VAR_IN_OUT
	awBusDataToVTEM 				: ARRAY [0..2] OF WORD; 	(* 6 bytes of process data sent to the Motion Terminal *)	
END_VAR

VAR_INPUT
	xExecute 						: BOOL; 					(* has to be set to TRUE for a download and to FALSE to reset the function block after a download *)
		                    		
	iParameterSet					: INT := 1; 				(* the parameter set to be written to, 1 by default *)
	
	// system parameters
		iTubingLengthAt2 			: INT; 						(* length of the tubing connected to outlet port 2 of the valve [1 digit = 1 mm] *)
		iTubingLengthAt4 			: INT;						(* length of the tubing connected to outlet port 4 of the valve [1 digit = 1 mm] *)
		iTubingInnerDiameterAt2 	: INT;  					(* inner diameter of the tubing connected to outlet port 2 of the valve [1 digit = 0.01 mm] *)
		iTubingInnerDiameterAt4 	: INT;						(* inner diameter of the tubing connected to outlet port 4 of the valve [1 digit = 0.01 mm] *)
		iVolumeAt2 					: INT; 						(* size/capacity of the volume connected to outlet port 2 of the valve [1 digit = 0.001 l] *)
	 	iVolumeAt4 					: INT;						(* size/capacity of the volume connected to outlet port 4 of the valve [1 digit = 0.001 l] *)
		iInPortRetracted_optional	: INT;						// Sensor port for detection of end position at pressurisation of outlet port 2 (retracted), value is number of the slot (beginning from 0) * 10 + number of the port
		iInPortAdvanced_optional	: INT;						// Sensor port for detection of end position at pressurisation of outlet port 4 (advanced), value is number of the slot (beginning from 0) * 10 + number of the port
    
	// application parameters
		iPressureRiseAt2 			: INT; 						(* maximum pressure rise at outlet port 2 [1 digit = 0.01 bar/s] *)
		iPressureRiseAt4 			: INT;						(* maximum pressure rise at outlet port 4 [1 digit = 0.01 bar/s] *)
END_VAR

VAR_OUTPUT
	iResponse 						: eTransferResponse; 		(* returns the status of the execution of the download process *)
	sCurrentValue 					: STRING; 					(* indicates which value of the array is currently treated (necessary to evaluate in case of error messages) *)
	xDownloadDone 					: BOOL; 					(* indicates whether the download was successful *)
	xDownloadError 					: BOOL := FALSE; 			(* indicates whether an error occurred during the transfer *)
END_VAR

VAR
	aTransferPackages				: ARRAY [0..100] OF stTransferPackage;
	fbdownloadMultipleParameters 	: FB_Download_Multiple_Parameters;
	iCurrentValue					: INT;
	fbWriteValueToWord 				: FB_Write_Value_To_Word;
END_VAR

(*****************************************************************************************************

Festo SE & Co. KG, Esslingen
Copyright (c) 2018. All rights reserved.

Product:            Motion Terminal VTEM
Description:        Function block to download the parameters for Motion App 4 to the Motion Terminal

Object version:     2.00
Last change:        2019-03
======================================================================================================
                                       H I S T O R Y
======================================================================================================
Version:            2.00
Date:               2019-03
Change/Activity:    - added parameters for the sensor port mapping (#2256294)
                    - changed awBusDataToVTEM into VAR_IN_OUT (#2368965)
Release:            3.5.7.230 (CODESYS 3.5.7.2, Lib version 3.0)
Author:             JEBU
------------------------------------------------------------------------------------------------------
Version:            1.00
Date:               2017
Change/Activity:    - created
Release:            3.5.7.220
Author:             HLBG
======================================================================================================

*****************************************************************************************************)

// write the Motion App specific parameters into the struct
	//iTubingLengthAt2
		aTransferPackages[0].iChannel := iParameterSet;
		aTransferPackages[0].iAddressedTarget := 4;
		aTransferPackages[0].iIndex := 12;
		aTransferPackages[0].iTransferValue := iTubingLengthAt2;
	
	//iTubingLengthAt4
		aTransferPackages[1].iChannel := iParameterSet;
		aTransferPackages[1].iAddressedTarget := 4;
		aTransferPackages[1].iIndex := 13;
		aTransferPackages[1].iTransferValue := iTubingLengthAt4;
	
	//iTubingInnerDiameterAt2
		aTransferPackages[2].iChannel := iParameterSet;
		aTransferPackages[2].iAddressedTarget := 4;
		aTransferPackages[2].iIndex := 14;
		aTransferPackages[2].iTransferValue := iTubingInnerDiameterAt2;
	
	//iTubingInnerDiameterAt4
		aTransferPackages[3].iChannel := iParameterSet;
		aTransferPackages[3].iAddressedTarget := 4;
		aTransferPackages[3].iIndex := 15;
		aTransferPackages[3].iTransferValue := iTubingInnerDiameterAt4;
	
	//iVolumeAt2
		aTransferPackages[4].iChannel := iParameterSet;
		aTransferPackages[4].iAddressedTarget := 4;
		aTransferPackages[4].iIndex := 40;
		aTransferPackages[4].iTransferValue := iVolumeAt2;
	
	//iVolumeAt4
		aTransferPackages[5].iChannel := iParameterSet;
		aTransferPackages[5].iAddressedTarget := 4;
		aTransferPackages[5].iIndex := 41;
		aTransferPackages[5].iTransferValue := iVolumeAt4;
	
	//iPressureRiseAt2
		aTransferPackages[6].iChannel := iParameterSet;
		aTransferPackages[6].iAddressedTarget := 4;
		aTransferPackages[6].iIndex := 182;
		aTransferPackages[6].iTransferValue := iPressureRiseAt2;
	
	//iPressureRiseAt4
		aTransferPackages[7].iChannel := iParameterSet;
		aTransferPackages[7].iAddressedTarget := 4;
		aTransferPackages[7].iIndex := 183;
		aTransferPackages[7].iTransferValue := iPressureRiseAt4;
	
	//iInPortRetract_optional
		aTransferPackages[8].iChannel := iParameterSet;
		aTransferPackages[8].iAddressedTarget := 4;
		aTransferPackages[8].iIndex := 70;
		aTransferPackages[8].iTransferValue := iInPortRetracted_optional;
	
	//iInPortAdvanced_optional
		aTransferPackages[9].iChannel := iParameterSet;
		aTransferPackages[9].iAddressedTarget := 4;
		aTransferPackages[9].iIndex := 71;
		aTransferPackages[9].iTransferValue := iInPortAdvanced_optional;
	
	// define end of parameter list to be downloaded by setting all variables to 0 (end criterion for FB_Download_Multiple_Parameters)
		aTransferPackages[10].iChannel := 0;
		aTransferPackages[10].iAddressedTarget := 0;
		aTransferPackages[10].iIndex := 0;
		aTransferPackages[10].iTransferValue := 0;


// pre-check of the value for the parameter set
	IF xExecute = TRUE AND (iParameterSet < 1 OR iParameterSet > 5) THEN		// invalid input for the parameter set
		xDownloadDone := FALSE; 
		xDownloadError := TRUE; 
		iResponse := eTransferResponse.invalid_ParameterSet; 
		iCurrentValue := 0; 
		// send command 'stop'
		fbWriteValueToWord(iValue := 61, iStartBit := 0, iEndBit := 5, wDataWord := awBusDataToVTEM[0]); 			// ValveMode = 61
		fbWriteValueToWord(iValue := 0, iStartBit := 6, iEndBit := 15, wDataWord := awBusDataToVTEM[0]); 			// (empty)
		awBusDataToVTEM[1] := 0; 
		awBusDataToVTEM[2] := 0; 
		
	ELSE	
		// call the function block for multiple parameter download
			fbdownloadMultipleParameters(	xExecute := xExecute,
											awBusDataFromVTEM := awBusDataFromVTEM,
											aTransferPackages := aTransferPackages, 
											awBusDataToVTEM := awBusDataToVTEM,
											xDownloadDone => xDownloadDone,
											xDownloadError => xDownloadError,
											iResponse => iResponse,
											iCurrentValue => iCurrentValue);
	END_IF
	

// The current value output is needed if there is any invalid value in order to address it correctly.
// As the user doesn't work with indices in this function block, the current value is transformed to a string holding the name of the parameter.
	CASE iCurrentValue OF
		0: sCurrentValue := 'iTubingLengthAt2';
		1: sCurrentValue := 'iTubingLengthAt4';
		2: sCurrentValue := 'iTubingInnerDiameterAt2';
		3: sCurrentValue := 'iTubingInnerDiameterAt4';
		4: sCurrentValue := 'iVolumeAt2';
		5: sCurrentValue := 'iVolumeAt4';
		6: sCurrentValue := 'iPressureRiseAt2';
		7: sCurrentValue := 'iPressureRiseAt4';
		8: sCurrentValue := 'iInPortRetract_optional';
		9: sCurrentValue := 'iInPortAdvanced_optional';
		10: sCurrentValue := 'AllParametersWritten';
	END_CASE

END_FUNCTION_BLOCK

// Transfermode/specific_MA_config/FB_Write_config_MA_11
/// This function block can be used to download the configuration of Motion App 11 ("Soft stop").
/// The specific parameters of this Motion App are the inputs of this FB and can be defined by the user. 
/// The function block uses the transfer mode to write this configuration to the Motion Terminal
/// and indicates the state of the download process.

FUNCTION_BLOCK FB_Write_config_MA_11
VAR_INPUT
	awBusDataFromVTEM 				: ARRAY [0..2] OF WORD;		(* 6 bytes of process data received from the Motion Terminal *)
END_VAR

VAR_IN_OUT
	awBusDataToVTEM					: ARRAY [0..2] OF WORD; 	(* 6 bytes of process data sent to the Motion Terminal *)
END_VAR

VAR_INPUT
	xExecute 						: BOOL; 					(* has to be set to TRUE for a download and to FALSE to reset the function block after a download *)
	
	iParameterSet					: INT := 1; 				(* the parameter set to be written to, 1 by default *)
	
	// system parameters
		iDriveType 					: INT;						(* type of the drive/cylinder/... that is to be operated by the valve ->  see list of drive types *)
	 	iDriveStroke 				: INT; 						(* stroke of the drive/cylinder/... that is to be operated by the valve [1 digit = 1 mm for linear drives, 1 digit = 1° for rotary drives] *)
		iInstallationPositionDrive 	: INT;  	 				(* inclination of the cylinder with reference to a horizontal installation position [1 digit = 0.01°, positive values = advancing upwards] *)
		iInPortRetracted			: INT;						// Sensor port for detection of end position at pressurisation of outlet port 2 (retracted), value is number of the slot (beginning from 0) * 10 + number of the port
		iInPortAdvanced				: INT;						// Sensor port for detection of end position at pressurisation of outlet port 4 (advanced), value is number of the slot (beginning from 0) * 10 + number of the port
	
	// application parameters                               	
	 	iLoadAdvancing 				: INT := 0; 				(* mass that is to be moved by the drive when advancing ((4) pressurised) [1 digit = 0.01 kg] *)
		iLoadRetracting 			: INT := 0;					(* mass that is to be moved by the drive when retracting ((2) pressurised) [1 digit = 0.01 kg] *)

END_VAR

VAR_OUTPUT                                                  	
	iResponse 						: eTransferResponse; 		(* returns the status of the execution of the download process *)
	sCurrentValue 					: STRING; 					(* indicates which value of the array is currently treated (necessary to evaluate in case of error messages) *)
	xDownloadDone 					: BOOL; 					(* indicates whether the download was successful *)
	xDownloadError 					: BOOL := FALSE; 			(* indicates whether an error occurred during the transfer *)
END_VAR

VAR
	aTransferPackages				: ARRAY [0..100] OF stTransferPackage;
	fbdownloadMultipleParameters 	: FB_Download_Multiple_Parameters;
	iCurrentValue					: INT;
	fbWriteValueToWord 				: FB_Write_Value_To_Word;
END_VAR

(*****************************************************************************************************

Festo SE & Co. KG, Esslingen
Copyright (c) 2018. All rights reserved.

Product:            Motion Terminal VTEM
Description:        Function block to download the parameters for Motion App 11 to the Motion Terminal

Object version:     2.01
Last change:        2019-03
======================================================================================================
                                       H I S T O R Y
======================================================================================================
Version:            2.01
Date:               2019-03
Change/Activity:    - sensor port mapping parameters (#2397241)
Release:            3.5.7.231 (CODESYS 3.5.7.2, Lib version 3.1)
Author:             JEBU
------------------------------------------------------------------------------------------------------
Version:            2.00
Date:               2019-03
Change/Activity:    - added parameters for the sensor port mapping (#2256294)
                    - removed tuning parameters (#2374189)
                    - changed awBusDataToVTEM into VAR_IN_OUT (#2368965)
Release:            3.5.7.230 (CODESYS 3.5.7.2, Lib version 3.0)
Author:             JEBU
------------------------------------------------------------------------------------------------------
Version:            1.01
Date:               2018-08
Change/Activity:    - added tuning parameters
Release:            3.5.7.220
Author:             JEBU
------------------------------------------------------------------------------------------------------
Version:            1.00
Date:               2017
Change/Activity:    - created
Release:            not released
Author:             HLBG
======================================================================================================

*****************************************************************************************************)

// write the Motion App specific parameters into the struct
	//iDriveType
		aTransferPackages[0].iChannel := iParameterSet;
		aTransferPackages[0].iAddressedTarget := 11;
		aTransferPackages[0].iIndex := 20;
		aTransferPackages[0].iTransferValue := iDriveType;
		
	//iDriveStroke
		aTransferPackages[1].iChannel := iParameterSet;
		aTransferPackages[1].iAddressedTarget := 11;
		aTransferPackages[1].iIndex := 21;
		aTransferPackages[1].iTransferValue := iDriveStroke;
		
	//iInstallationPositionDrive
		aTransferPackages[2].iChannel := iParameterSet;
		aTransferPackages[2].iAddressedTarget := 11;
		aTransferPackages[2].iIndex := 60;
		aTransferPackages[2].iTransferValue := iInstallationPositionDrive;
		
	//iLoadAdvancing
		aTransferPackages[3].iChannel := iParameterSet;
		aTransferPackages[3].iAddressedTarget := 11;
		aTransferPackages[3].iIndex := 101;
		aTransferPackages[3].iTransferValue := iLoadAdvancing;
		
	//iLoadRetracting
		aTransferPackages[4].iChannel := iParameterSet;
		aTransferPackages[4].iAddressedTarget := 11;
		aTransferPackages[4].iIndex := 100;
		aTransferPackages[4].iTransferValue := iLoadRetracting;
		
	//iInPortRetract
		aTransferPackages[5].iChannel := iParameterSet;
		aTransferPackages[5].iAddressedTarget := 11;
		aTransferPackages[5].iIndex := 75;
		aTransferPackages[5].iTransferValue := iInPortRetracted;
	
	//iInPortRetract
		aTransferPackages[6].iChannel := iParameterSet;
		aTransferPackages[6].iAddressedTarget := 11;
		aTransferPackages[6].iIndex := 76;
		aTransferPackages[6].iTransferValue := iInPortAdvanced;
	
	// define end of parameter list to be downloaded by setting all variables to 0 (end criterion for FB_Download_Multiple_Parameters)
		aTransferPackages[7].iChannel := 0;
		aTransferPackages[7].iAddressedTarget := 0;
		aTransferPackages[7].iIndex := 0;
		aTransferPackages[7].iTransferValue := 0;


// pre-check of the value for the parameter set
	IF xExecute = TRUE AND (iParameterSet < 1 OR iParameterSet > 5) THEN		// invalid input for the parameter set
		xDownloadDone := FALSE; 
		xDownloadError := TRUE; 
		iResponse := eTransferResponse.invalid_ParameterSet; 
		iCurrentValue := 0; 
		// send command 'stop'
		fbWriteValueToWord(iValue := 61, iStartBit := 0, iEndBit := 5, wDataWord := awBusDataToVTEM[0]); 			// ValveMode = 61
		fbWriteValueToWord(iValue := 0, iStartBit := 6, iEndBit := 15, wDataWord := awBusDataToVTEM[0]); 			// (empty)
		awBusDataToVTEM[1] := 0; 
		awBusDataToVTEM[2] := 0; 
		
	ELSE	
		// call the function block for multiple parameter download
			fbdownloadMultipleParameters(	xExecute := xExecute,
											awBusDataFromVTEM := awBusDataFromVTEM,
											aTransferPackages := aTransferPackages, 
											awBusDataToVTEM := awBusDataToVTEM,
											xDownloadDone => xDownloadDone,
											xDownloadError => xDownloadError,
											iResponse => iResponse,
											iCurrentValue => iCurrentValue);
	END_IF
		
	
// The current value output is needed if there is any invalid value in order to address it correctly.
// As the user doesn't work with indices in this function block, the current value is transformed to a string holding the name of the parameter.
	CASE iCurrentValue OF
		0: sCurrentValue := 'iDriveType';
		1: sCurrentValue := 'iDriveStroke';
		2: sCurrentValue := 'iInstallationPositionDrive';
		3: sCurrentValue := 'iLoadAdvancing';
		4: sCurrentValue := 'iLoadRetracting';
		5: sCurrentValue := 'iInPortRetract';
		6: sCurrentValue := 'iInPortAdvanced';
		7: sCurrentValue := 'AllParametersWritten';
	END_CASE

END_FUNCTION_BLOCK

// Transfermode/specific_MA_config/FB_Write_config_MA_12
/// This function block can be used to download the configuration of Motion App 12 ("Leakage diagnostics").
/// The specific parameters of this Motion App are the inputs of this FB and can be defined by the user. 
/// The function block uses the transfer mode to write this configuration to the Motion Terminal
/// and indicates the state of the download process.

FUNCTION_BLOCK FB_Write_config_MA_12
VAR_INPUT
	awBusDataFromVTEM 				: ARRAY [0..2] OF WORD;		(* 6 bytes of process data received from the Motion Terminal *)
END_VAR

VAR_IN_OUT
	awBusDataToVTEM 				: ARRAY [0..2] OF WORD; 	(* 6 bytes of process data sent to the Motion Terminal *)
END_VAR

VAR_INPUT
	xExecute 						: BOOL; 					(* has to be set to TRUE for a download and to FALSE to reset the function block after a download *)
		                                                    	
	iParameterSet					: INT := 1; 				(* the parameter set to be written to, 1 by default *)
	
	// system parameters
		iTubingLengthAt2 			: INT; 						(* length of the tubing connected to outlet port 2 of the valve [1 digit = 1 mm] *)
	 	iTubingLengthAt4 			: INT;						(* length of the tubing connected to outlet port 4 of the valve [1 digit = 1 mm] *)
	 	iTubingInnerDiameterAt2		: INT;  					(* inner diameter of the tubing connected to outlet port 2 of the valve [1 digit = 0.01mm] *)
	 	iTubingInnerDiameterAt4		: INT;						(* inner diameter of the tubing connected to outlet port 4 of the valve [1 digit = 0.01mm] *)
	 	iDriveType 					: INT;						(* type of the drive/cylinder/... that is to be operated by the valve ->  see list of drive types *)
	 	iDriveStroke 				: INT; 						(* stroke of the drive/cylinder/... that is to be operated by the valve [1 digit = 1 mm for linear drives, 1 digit = 1° for rotary drives] *)
		iVolumeAt2 					: INT; 						(* size/capacity of the volume connected to outlet port 2 of the valve [1 digit = 0.001 l] *)
		iVolumeAt4 					: INT;						(* size/capacity of the volume connected to outlet port 4 of the valve [1 digit = 0.001 l] *)
		iInstallationPositionDrive 	: INT;  	 				(* inclination of the cylinder with reference to a horizontal installation position [1 digit = 0.01°, positive values = advancing upwards] *)

	// application parameters                               	
		iLoadRetracting 			: INT;						(* mass that is to be moved by the drive when retracting ((2) pressurised) [1 digit = 0.01 kg] *)
	 	iLoadAdvancing 				: INT; 						(* mass that is to be moved by the drive when advancing ((4) pressurised) [1 digit = 0.01 kg] *)
		iMomentOfInertiaRetracting	: INT;						// Moment of inertia during for swivel drives when retratcting ((2) pressirised) [1 digit = 1 kg cm³]
		iMomentOfInertiaAdvancing	: INT;						// Moment of inertia during for swivel drives when advancing ((4) pressirised) [1 digit = 1 kg cm³]
		iMaxLeakageForStatusGood 	: INT;						(* allowed deviation regarding reference value for status "Good" [1 digit = 0.1 l/h] *)
		iMaxLeakageForStatusWarning : INT;						(* allowed deviation regarding reference value for status "Warning" [1 digit = 0.1 l/h] *)
	 	iMaxLeakageForStatusCritical: INT; 						(* allowed deviation regarding reference value for status "Critical" [1 digit = 0.1 l/h] *)
END_VAR

VAR_OUTPUT                                                  	
	iResponse 						: eTransferResponse;		(* returns the status of the execution of the download process *)
	sCurrentValue 					: STRING; 					(* indicates which value of the array is currently treated (necessary to evaluate in case of error messages) *)
	xDownloadDone 					: BOOL; 					(* indicates whether the download was successful *)
	xDownloadError 					: BOOL := FALSE; 			(* indicates whether an error occurred during the transfer *)
END_VAR

VAR
	aTransferPackages				: ARRAY [0..100] OF stTransferPackage;
	fbdownloadMultipleParameters 	: FB_Download_Multiple_Parameters;
	iCurrentValue					: INT;
	fbWriteValueToWord 				: FB_Write_Value_To_Word;
END_VAR

(*****************************************************************************************************

Festo SE & Co. KG, Esslingen
Copyright (c) 2018. All rights reserved.

Product:            Motion Terminal VTEM
Description:        Function block to download the parameters for Motion App 12 to the Motion Terminal

Object version:     2.01
Last change:        2019-04
======================================================================================================
                                       H I S T O R Y
======================================================================================================
Version:            2.01
Date:               2019-04
Change/Activity:    - added parameters for moment of inertia used for swivel drives (#2307852)
                    - changed awBusDataToVTEM into VAR_IN_OUT (#2368965)
Release:            3.5.7.231 (CODESYS 3.5.7.2, Lib version 3.1)
Author:             JEBU
------------------------------------------------------------------------------------------------------
Version:            1.00
Date:               2017
Change/Activity:    - created
Release:            3.5.7.22 (CODESYS 3.5.7.2, Lib version 2.0)
Author:             HLBG
======================================================================================================

*****************************************************************************************************)

// write the Motion App specific parameters into the struct
	//iTubingLengthAt2
		aTransferPackages[0].iChannel := iParameterSet;
		aTransferPackages[0].iAddressedTarget := 12;
		aTransferPackages[0].iIndex := 12;
		aTransferPackages[0].iTransferValue := iTubingLengthAt2;
		
	//iTubingLengthAt4
		aTransferPackages[1].iChannel := iParameterSet;
		aTransferPackages[1].iAddressedTarget := 12;
		aTransferPackages[1].iIndex := 13;
		aTransferPackages[1].iTransferValue := iTubingLengthAt4;
		
	//iTubingInnerDiameterAt2
		aTransferPackages[2].iChannel := iParameterSet;
		aTransferPackages[2].iAddressedTarget := 12;
		aTransferPackages[2].iIndex := 14;
		aTransferPackages[2].iTransferValue := iTubingInnerDiameterAt2;
		
	//iTubingInnerDiameterAt4
		aTransferPackages[3].iChannel := iParameterSet;
		aTransferPackages[3].iAddressedTarget := 12;
		aTransferPackages[3].iIndex := 15;
		aTransferPackages[3].iTransferValue := iTubingInnerDiameterAt4;
		
	//iDriveType
		aTransferPackages[4].iChannel := iParameterSet;
		aTransferPackages[4].iAddressedTarget := 12;
		aTransferPackages[4].iIndex := 20;
		aTransferPackages[4].iTransferValue := iDriveType;
		
	//iDriveStroke
		aTransferPackages[5].iChannel := iParameterSet;
		aTransferPackages[5].iAddressedTarget := 12;
		aTransferPackages[5].iIndex := 21;
		aTransferPackages[5].iTransferValue := iDriveStroke;
		
	//iVolumeAt2
		aTransferPackages[6].iChannel := iParameterSet;
		aTransferPackages[6].iAddressedTarget := 12;
		aTransferPackages[6].iIndex := 40;
		aTransferPackages[6].iTransferValue := iVolumeAt2;
		
	//iVolumeAt4 
		aTransferPackages[7].iChannel := iParameterSet;
		aTransferPackages[7].iAddressedTarget := 12;
		aTransferPackages[7].iIndex := 41;
		aTransferPackages[7].iTransferValue := iVolumeAt4;
		
	//iInstallationPositionDrive
		aTransferPackages[8].iChannel := iParameterSet;
		aTransferPackages[8].iAddressedTarget := 12;
		aTransferPackages[8].iIndex := 60;
		aTransferPackages[8].iTransferValue := iInstallationPositionDrive;
		
	//iLoadRetracting
		aTransferPackages[9].iChannel := iParameterSet;
		aTransferPackages[9].iAddressedTarget := 12;
		aTransferPackages[9].iIndex := 100;
		aTransferPackages[9].iTransferValue := iLoadRetracting;
		
	//iLoadAdvancing
		aTransferPackages[10].iChannel := iParameterSet;
		aTransferPackages[10].iAddressedTarget := 12;
		aTransferPackages[10].iIndex := 101;
		aTransferPackages[10].iTransferValue := iLoadAdvancing;
		
	//iMomentOfInertiaRetracting
		aTransferPackages[11].iChannel := iParameterSet;
		aTransferPackages[11].iAddressedTarget := 12;
		aTransferPackages[11].iIndex := 102;
		aTransferPackages[11].iTransferValue := iMomentOfInertiaRetracting;
	
	//iMomentOfInertiaAdvancing
		aTransferPackages[12].iChannel := iParameterSet;
		aTransferPackages[12].iAddressedTarget := 12;
		aTransferPackages[12].iIndex := 103;
		aTransferPackages[12].iTransferValue := iMomentOfInertiaAdvancing;

	//iMaxLeakageForStatusGood
		aTransferPackages[13].iChannel := iParameterSet;
		aTransferPackages[13].iAddressedTarget := 12;
		aTransferPackages[13].iIndex := 200;
		aTransferPackages[13].iTransferValue := iMaxLeakageForStatusGood;
		
	//iMaxLeakageForStatusWarning
		aTransferPackages[14].iChannel := iParameterSet;
		aTransferPackages[14].iAddressedTarget := 12;
		aTransferPackages[14].iIndex := 201;
		aTransferPackages[14].iTransferValue := iMaxLeakageForStatusWarning;
		
	//iMaxLeakageForStatusCritical
		aTransferPackages[15].iChannel := iParameterSet;
		aTransferPackages[15].iAddressedTarget := 12;
		aTransferPackages[15].iIndex := 202;
		aTransferPackages[15].iTransferValue := iMaxLeakageForStatusCritical;
	
	// define end of parameter list to be downloaded by setting all variables to 0 (end criterion for FB_Download_Multiple_Parameters)
		aTransferPackages[16].iChannel := 0;
		aTransferPackages[16].iAddressedTarget := 0;
		aTransferPackages[16].iIndex := 0;
		aTransferPackages[16].iTransferValue := 0;


// pre-check of the value for the parameter set
	IF xExecute = TRUE AND (iParameterSet < 1 OR iParameterSet > 5) THEN		// invalid input for the parameter set
		xDownloadDone := FALSE; 
		xDownloadError := TRUE; 
		iResponse := eTransferResponse.invalid_ParameterSet; 
		iCurrentValue := 0; 
		// send command 'stop'
		fbWriteValueToWord(iValue := 61, iStartBit := 0, iEndBit := 5, wDataWord := awBusDataToVTEM[0]); 			// ValveMode = 61
		fbWriteValueToWord(iValue := 0, iStartBit := 6, iEndBit := 15, wDataWord := awBusDataToVTEM[0]); 			// (empty)
		awBusDataToVTEM[1] := 0; 
		awBusDataToVTEM[2] := 0; 
		
	ELSE	
		// call the function block for multiple parameter download
			fbdownloadMultipleParameters(	xExecute := xExecute,
											awBusDataFromVTEM := awBusDataFromVTEM,
											aTransferPackages := aTransferPackages, 
											awBusDataToVTEM := awBusDataToVTEM,
											xDownloadDone => xDownloadDone,
											xDownloadError => xDownloadError,
											iResponse => iResponse,
											iCurrentValue => iCurrentValue);
	END_IF
		
	
// The current value output is needed if there is any invalid value in order to address it correctly.
// As the user doesn't work with indices in this function block, the current value is transformed to a string holding the name of the parameter.
	CASE iCurrentValue OF
		0: sCurrentValue := 'iTubingLengthAt2';
		1: sCurrentValue := 'iTubingLengthAt4';
		2: sCurrentValue := 'iTubingInnerDiameterAt2';
		3: sCurrentValue := 'iTubingInnerDiameterAt4';
		4: sCurrentValue := 'iDriveType';
		5: sCurrentValue := 'iDriveStroke';
		6: sCurrentValue := 'iVolumeAt2';
		7: sCurrentValue := 'iVolumeAt4';
		8: sCurrentValue := 'iInstallationPositionDrive';
		9: sCurrentValue := 'iLoadRetracting';
		10: sCurrentValue := 'iLoadAdvancing';
		11: sCurrentValue := 'iMomentOfInertiaRetracting';
		12: sCurrentValue := 'iMomentOfInertiaAdvancing';
		13: sCurrentValue := 'iMaxLeakageForStatusGood';
		14: sCurrentValue := 'iMaxLeakageForStatusWarning';
		15: sCurrentValue := 'iMaxLeakageForStatusCritical';
		16: sCurrentValue := 'AllParametersWritten';
	END_CASE

END_FUNCTION_BLOCK

// StateInterpreter/FB_StateInterpreter_MA_02
/// The variable "byActualAppState" is an output of the FB_ValveControl that is used differently in each Motion App.
/// This function block interprets the "AppState" output of the FB_ValveControl if Motion App 2 ("Proportional directional control valve") is running.
/// The Motion App specific values are derived from the "byActualAppState".

FUNCTION_BLOCK FB_StateInterpreter_MA_02
VAR_INPUT
	byActualAppState 			: BYTE; 	(* output of the FB_ValveControl *)
END_VAR
VAR_OUTPUT
	xRetractedEndPos_optional	: BOOL;  	(* only if digital sensors are installed (optional): indicates whether the retracted end position was reached (after outlet port 2 is pressurised) *)
	xAdvancedEndPos_optional	: BOOL;  	(* only if digital sensors are installed (optional): indicates whether the advanced end position was reached (after outlet port 4 is pressurised) *)
	xWarning					: BOOL; 	(* indicates whether there is a warning returned by the Motion App *)
END_VAR
VAR
	fbReadBitsFromByte			: FB_Read_Bits_From_Byte;
	byRetractedEndPos			: BYTE;
	byAdvancedEndPos			: BYTE;
	byWarning					: BYTE;
END_VAR

(*****************************************************************************************************

Festo SE & Co. KG, Esslingen
Copyright (c) 2018. All rights reserved.

Product:            Motion Terminal VTEM
Description:        Function block for interpreting the app state of Motion App 2

Object version:     1.00
Last change:        2017
======================================================================================================
                                       H I S T O R Y
======================================================================================================
Version:            1.00
Date:               2017
Change/Activity:    - created
Release:            3.5.7.220
Author:             HLBG
======================================================================================================

*****************************************************************************************************)

// read the Motion App specific values from the ActualAppState byte
fbReadBitsFromByte(byData := byActualAppState, iStartBit := 0, iEndBit := 0, byValue => byRetractedEndPos);
xRetractedEndPos_optional :=  BYTE_TO_BIT(byRetractedEndPos);

fbReadBitsFromByte(byData := byActualAppState, iStartBit := 2, iEndBit := 2, byValue => byAdvancedEndPos); 
xAdvancedEndPos_optional :=  BYTE_TO_BIT(byAdvancedEndPos);

fbReadBitsFromByte(byData := byActualAppState, iStartBit := 7, iEndBit := 7, byValue => byWarning);
xWarning := BYTE_TO_BIT(byWarning);

END_FUNCTION_BLOCK

// StateInterpreter/FB_StateInterpreter_MA_03
/// The variable "byActualAppState" is an output of the FB_ValveControl that is used differently in each Motion App.
/// This function block interprets the "AppState" output of the FB_ValveControl if Motion App 3 ("Proportional pressure regulation") is running.
/// The Motion App specific values are derived from the "byActualAppState".

FUNCTION_BLOCK FB_StateInterpreter_MA_03
VAR_INPUT
	byActualAppState 			: BYTE; 	(* output of the FB_ValveControl *)
END_VAR
VAR_OUTPUT
	xRetractedEndPos_optional	: BOOL;  	(* only if digital sensors are installed (optional): indicates whether the retracted end position was reached (after outlet port 2 is pressurised) *)
	xAdvancedEndPos_optional	: BOOL;  	(* only if digital sensors are installed (optional): indicates whether the advanced end position was reached (after outlet port 4 is pressurised) *)
	xWarning					: BOOL; 	(* indicates whether there is a warning returned by the Motion App *)
END_VAR
VAR
	fbReadBitsFromByte			: FB_Read_Bits_From_Byte;
	byRetractedEndPos			: BYTE;
	byAdvancedEndPos			: BYTE;
	byWarning					: BYTE;
END_VAR

(*****************************************************************************************************

Festo SE & Co. KG, Esslingen
Copyright (c) 2018. All rights reserved.

Product:            Motion Terminal VTEM
Description:        Function block for interpreting the app state of Motion App 3

Object version:     1.00
Last change:        2017
======================================================================================================
                                       H I S T O R Y
======================================================================================================
Version:            1.00
Date:               2017
Change/Activity:    - created
Release:            3.5.7.220
Author:             HLBG
======================================================================================================

*****************************************************************************************************)

// read the Motion App specific values from the ActualAppState byte
fbReadBitsFromByte(byData := byActualAppState, iStartBit := 0, iEndBit := 0, byValue => byRetractedEndPos);
xRetractedEndPos_optional :=  BYTE_TO_BIT(byRetractedEndPos);

fbReadBitsFromByte(byData := byActualAppState, iStartBit := 2, iEndBit := 2, byValue => byAdvancedEndPos); 
xAdvancedEndPos_optional :=  BYTE_TO_BIT(byAdvancedEndPos);

fbReadBitsFromByte(byData := byActualAppState, iStartBit := 7, iEndBit := 7, byValue => byWarning);
xWarning := BYTE_TO_BIT(byWarning);

END_FUNCTION_BLOCK

// StateInterpreter/FB_StateInterpreter_MA_04
/// The variable "byActualAppState" is an output of the FB_ValveControl that is used differently in each Motion App.
/// This function block interprets the "AppState" output of the FB_ValveControl if Motion App 4 ("Model-based proportional pressure regulation") is running.
/// The Motion App specific values are derived from the "byActualAppState".

FUNCTION_BLOCK FB_StateInterpreter_MA_04
VAR_INPUT
	byActualAppState 			: BYTE; 	(* output of the FB_ValveControl *)
END_VAR
VAR_OUTPUT
	xRetractedEndPos_optional	: BOOL;  	(* only if digital sensors are installed (optional): indicates whether the retracted end position was reached (after outlet port 2 is pressurised) *)
	xAdvancedEndPos_optional	: BOOL;  	(* only if digital sensors are installed (optional): indicates whether the advanced end position was reached (after outlet port 4 is pressurised) *)
	xWarning					: BOOL; 	(* indicates whether there is a warning returned by the Motion App *)
END_VAR
VAR
	fbReadBitsFromByte			: FB_Read_Bits_From_Byte;
	byRetractedEndPos			: BYTE;
	byAdvancedEndPos			: BYTE;
	byWarning					: BYTE;
END_VAR

(*****************************************************************************************************

Festo SE & Co. KG, Esslingen
Copyright (c) 2018. All rights reserved.

Product:            Motion Terminal VTEM
Description:        Function block for interpreting the app state of Motion App 4

Object version:     1.00
Last change:        2017
======================================================================================================
                                       H I S T O R Y
======================================================================================================
Version:            1.00
Date:               2017
Change/Activity:    - created
Release:            3.5.7.220
Author:             HLBG
======================================================================================================

*****************************************************************************************************)

// read the Motion App specific values from the ActualAppState byte
fbReadBitsFromByte(byData := byActualAppState, iStartBit := 0, iEndBit := 0, byValue => byRetractedEndPos);
xRetractedEndPos_optional :=  BYTE_TO_BIT(byRetractedEndPos);

fbReadBitsFromByte(byData := byActualAppState, iStartBit := 2, iEndBit := 2, byValue => byAdvancedEndPos); 
xAdvancedEndPos_optional :=  BYTE_TO_BIT(byAdvancedEndPos);

fbReadBitsFromByte(byData := byActualAppState, iStartBit := 7, iEndBit := 7, byValue => byWarning);
xWarning := BYTE_TO_BIT(byWarning);

END_FUNCTION_BLOCK

// StateInterpreter/FB_StateInterpreter_MA_05
/// The variable "byActualAppState" is an output of the FB_ValveControl that is used differently in each Motion App.
/// This function block interprets the "AppState" output of the FB_ValveControl if Motion App 5 ("Supply and exhaust air flow control") is running.
/// The Motion App specific values are derived from the "byActualAppState".

FUNCTION_BLOCK FB_StateInterpreter_MA_05
VAR_INPUT
	byActualAppState 			: BYTE; 	(* output of the FB_ValveControl *)
END_VAR
VAR_OUTPUT
	xRetractedEndPos_optional	: BOOL;  	(* only if digital sensors are installed (optional): indicates whether the retracted end position was reached (after outlet port 2 is pressurised) *)
	xAdvancedEndPos_optional	: BOOL;  	(* only if digital sensors are installed (optional): indicates whether the advanced end position was reached (after outlet port 4 is pressurised) *)
	xWarning					: BOOL; 	(* indicates whether there is a warning returned by the Motion App *)
END_VAR
VAR
	fbReadBitsFromByte			: FB_Read_Bits_From_Byte;
	byRetractedEndPos			: BYTE;
	byAdvancedEndPos			: BYTE;
	byWarning					: BYTE;
END_VAR

(*****************************************************************************************************

Festo SE & Co. KG, Esslingen
Copyright (c) 2018. All rights reserved.

Product:            Motion Terminal VTEM
Description:        Function block for interpreting the app state of Motion App 5 

Object version:     1.00
Last change:        2017
======================================================================================================
                                       H I S T O R Y
======================================================================================================
Version:            1.00
Date:               2017
Change/Activity:    - created
Release:            3.5.7.220
Author:             HLBG
======================================================================================================

*****************************************************************************************************)

// read the Motion App specific values from the ActualAppState byte
fbReadBitsFromByte(byData := byActualAppState, iStartBit := 0, iEndBit := 0, byValue => byRetractedEndPos);
xRetractedEndPos_optional :=  BYTE_TO_BIT(byRetractedEndPos);

fbReadBitsFromByte(byData := byActualAppState, iStartBit := 2, iEndBit := 2, byValue => byAdvancedEndPos); 
xAdvancedEndPos_optional :=  BYTE_TO_BIT(byAdvancedEndPos);

fbReadBitsFromByte(byData := byActualAppState, iStartBit := 7, iEndBit := 7, byValue => byWarning);
xWarning := BYTE_TO_BIT(byWarning);

END_FUNCTION_BLOCK

// StateInterpreter/FB_StateInterpreter_MA_08
/// The variable "byActualAppState" is an output of the FB_ValveControl that is used differently in each Motion App.
/// This function block interprets the "AppState" output of the FB_ValveControl if Motion App 8 ("Selectable pressure level (ECO)") is running.
/// The Motion App specific values are derived from the "byActualAppState".

FUNCTION_BLOCK FB_StateInterpreter_MA_08
VAR_INPUT
	byActualAppState 			: BYTE; 	(* output of the FB_ValveControl *)
END_VAR
VAR_OUTPUT
	xRetractedEndPos_optional	: BOOL;  	(* only if digital sensors are installed (optional): indicates whether the retracted end position was reached (after outlet port 2 is pressurised) *)
	xAdvancedEndPos_optional	: BOOL;  	(* only if digital sensors are installed (optional): indicates whether the advanced end position was reached (after outlet port 4 is pressurised) *)
	xWarning					: BOOL; 	(* indicates whether there is a warning returned by the Motion App *)
END_VAR
VAR
	fbReadBitsFromByte			: FB_Read_Bits_From_Byte;
	byRetractedEndPos			: BYTE;
	byAdvancedEndPos			: BYTE;
	byWarning					: BYTE;
END_VAR

(*****************************************************************************************************

Festo SE & Co. KG, Esslingen
Copyright (c) 2018. All rights reserved.

Product:            Motion Terminal VTEM
Description:        Function block for interpreting the app state of Motion App 8 

Object version:     1.00
Last change:        2017
======================================================================================================
                                       H I S T O R Y
======================================================================================================
Version:            1.00
Date:               2017
Change/Activity:    - created
Release:            3.5.7.220
Author:             HLBG
======================================================================================================

*****************************************************************************************************)

// read the Motion App specific values from the ActualAppState byte
fbReadBitsFromByte(byData := byActualAppState, iStartBit := 0, iEndBit := 0, byValue => byRetractedEndPos);
xRetractedEndPos_optional :=  BYTE_TO_BIT(byRetractedEndPos);

fbReadBitsFromByte(byData := byActualAppState, iStartBit := 2, iEndBit := 2, byValue => byAdvancedEndPos); 
xAdvancedEndPos_optional :=  BYTE_TO_BIT(byAdvancedEndPos);

fbReadBitsFromByte(byData := byActualAppState, iStartBit := 7, iEndBit := 7, byValue => byWarning);
xWarning := BYTE_TO_BIT(byWarning);

END_FUNCTION_BLOCK

// Transfermode/specific_MA_config/FB_Write_config_MA_02
/// This function block can be used to download the configuration of Motion App 2 ("Proportional directional control valve").
/// The specific parameters of this Motion App are the inputs of this FB and can be defined by the user. 
/// The function block uses the transfer mode to write this configuration to the Motion Terminal
/// and indicates the state of the download process.

FUNCTION_BLOCK FB_Write_config_MA_02
VAR_INPUT
	awBusDataFromVTEM 				: ARRAY [0..2] OF WORD;		(* 6 bytes of process data received from the Motion Terminal *)
END_VAR

VAR_IN_OUT
	awBusDataToVTEM 				: ARRAY [0..2] OF WORD; 	(* 6 bytes of process data sent to the Motion Terminal *)
END_VAR
		
VAR_INPUT
	xExecute 						: BOOL; 					(* has to be set to TRUE for a download and to FALSE to reset the function block after a download *)

	iParameterSet					: INT := 1; 				(* the parameter set to be written to, 1 by default *)

	// system parameters
		iInPortRetracted_optional	: INT;						// Sensor port for detection of end position at pressurisation of outlet port 2 (retracted), value is number of the slot (beginning from 0) * 10 + number of the port
		iInPortAdvanced_optional	: INT;						// Sensor port for detection of end position at pressurisation of outlet port 4 (advanced), value is number of the slot (beginning from 0) * 10 + number of the port
	
	// application parameters
		iCharacteristicAt2 			: INT := 0; 			(* characteristic of the control algorithm for outlet port 2 -> choose characteristic from list *)
		iCharacteristicAt4 			: INT := 0; 			(* characteristic of the control algorithm for outlet port 4 -> choose characteristic from list *)
END_VAR                     		

VAR_OUTPUT                  		
	iResponse 						: eTransferResponse; 		(* returns the status of the execution of the download process *)
	sCurrentValue 					: STRING; 					(* indicates which value of the array is currently treated (necessary to evaluate in case of error messages) *)
	xDownloadDone 					: BOOL; 					(* indicates whether the download was successful *)
	xDownloadError 					: BOOL := FALSE; 			(* indicates whether an error occurred during the transfer *)
END_VAR

VAR
	aTransferPackages				: ARRAY [0..100] OF stTransferPackage;
	fbdownloadMultipleParameters	: FB_Download_Multiple_Parameters;
	iCurrentValue					: INT;
	fbWriteValueToWord 				: FB_Write_Value_To_Word;
END_VAR

(*****************************************************************************************************

Festo SE & Co. KG, Esslingen
Copyright (c) 2018. All rights reserved.

Product:            Motion Terminal VTEM
Description:        Function block to download the parameters for Motion App 2 to the Motion Terminal

Object version:     2.00
Last change:        2019-03
======================================================================================================
                                       H I S T O R Y
======================================================================================================
Version:            2.00
Date:               2019-03
Change/Activity:    - added parameters for the sensor port mapping (#2256294)
					- changed awBusDataToVTEM into VAR_IN_OUT (#2368965)
Release:            3.5.7.230 (CODESYS 3.5.7.2, Lib version 3.0)
Author:             JEBU
======================================================================================================
Version:            1.00
Date:               2017
Change/Activity:    - created
Release:            3.5.7.220
Author:             HLBG
======================================================================================================

*****************************************************************************************************)

// write the Motion App specific parameters into the struct
	//iCharacteristicAt2
		aTransferPackages[0].iChannel := iParameterSet;
		aTransferPackages[0].iAddressedTarget := 2;
		aTransferPackages[0].iIndex := 220;
		aTransferPackages[0].iTransferValue := iCharacteristicAt2;
	
	//iCharacteristicAt4
		aTransferPackages[1].iChannel := iParameterSet;
		aTransferPackages[1].iAddressedTarget := 2;
		aTransferPackages[1].iIndex := 221;
		aTransferPackages[1].iTransferValue := iCharacteristicAt4;
	
	//iInPortRetract_optional
		aTransferPackages[2].iChannel := iParameterSet;
		aTransferPackages[2].iAddressedTarget := 2;
		aTransferPackages[2].iIndex := 70;
		aTransferPackages[2].iTransferValue := iInPortRetracted_optional;
	
	//iInPortAdvanced_optional
		aTransferPackages[3].iChannel := iParameterSet;
		aTransferPackages[3].iAddressedTarget := 2;
		aTransferPackages[3].iIndex := 71;
		aTransferPackages[3].iTransferValue := iInPortAdvanced_optional;
	
	// define end of parameter list to be downloaded by setting all variables to 0 (end criterion for FB_Download_Multiple_Parameters)
		aTransferPackages[4].iChannel := 0;
		aTransferPackages[4].iAddressedTarget := 0;
		aTransferPackages[4].iIndex := 0;
		aTransferPackages[4].iTransferValue := 0;


// pre-check of the value for the parameter set
	IF xExecute = TRUE AND (iParameterSet < 1 OR iParameterSet > 5) THEN		// invalid input for the parameter set
		xDownloadDone := FALSE; 
		xDownloadError := TRUE; 
		iResponse := eTransferResponse.invalid_ParameterSet; 
		iCurrentValue := 0; 
		// send command 'stop'
		fbWriteValueToWord(iValue := 61, iStartBit := 0, iEndBit := 5, wDataWord := awBusDataToVTEM[0]); 			// ValveMode = 61
		fbWriteValueToWord(iValue := 0, iStartBit := 6, iEndBit := 15, wDataWord := awBusDataToVTEM[0]); 			// (empty)
		awBusDataToVTEM[1] := 0; 
		awBusDataToVTEM[2] := 0; 
		
	ELSE	
		// call the function block for multiple parameter download
		fbdownloadMultipleParameters(	xExecute := xExecute,
										awBusDataFromVTEM := awBusDataFromVTEM,
										aTransferPackages := aTransferPackages, 
										awBusDataToVTEM := awBusDataToVTEM,
										xDownloadDone => xDownloadDone,
										xDownloadError => xDownloadError,
										iResponse => iResponse,
										iCurrentValue => iCurrentValue);
	END_IF


// The current value output is needed if there is any invalid value in order to address it correctly.
// As the user doesn't work with indices in this function block, the current value is transformed to a string holding the name of the parameter.
	CASE iCurrentValue OF
		0: sCurrentValue := 'iCharacteristicAt2';
		1: sCurrentValue := 'iCharacteristicAt4';
		2: sCurrentValue := 'iInPortRetract_optional';
		3: sCurrentValue := 'iInPortAdvanced_optional';
		4: sCurrentValue := 'AllParametersWritten';
	END_CASE

END_FUNCTION_BLOCK

// Transfermode/specific_MA_config/FB_Write_config_MA_03
/// This function block can be used to download the configuration of Motion App 3 ("Proportional pressure regulation").
/// The specific parameters of this Motion App are the inputs of this FB and can be defined by the user. 
/// The function block uses the transfer mode to write this configuration to the Motion Terminal
/// and indicates the state of the download process.

FUNCTION_BLOCK FB_Write_config_MA_03
VAR_INPUT
	awBusDataFromVTEM 				: ARRAY [0..2] OF WORD;		(* 6 bytes of process data received from the Motion Terminal *)
END_VAR	

VAR_IN_OUT
	awBusDataToVTEM 				: ARRAY [0..2] OF WORD; 	(* 6 bytes of process data sent to the Motion Terminal *)
END_VAR

VAR_INPUT
	xExecute 						: BOOL; 					(* has to be set to TRUE for a download and to FALSE to reset the function block after a download *)
		                    		
	iParameterSet					: INT := 1; 				(* the parameter set to be written to, 1 by default *)
	
	// system parameters
		iInPortRetracted_optional	: INT;						// Sensor port for detection of end position at pressurisation of outlet port 2 (retracted), value is number of the slot (beginning from 0) * 10 + number of the port
		iInPortAdvanced_optional	: INT;						// Sensor port for detection of end position at pressurisation of outlet port 4 (advanced), value is number of the slot (beginning from 0) * 10 + number of the port
	
	// application parameters
		iCharacteristicAt2 			: INT;		 				(* characteristic of the control algorithm for outlet port 2 -> choose characteristic from list *)
		iCharacteristicAt4 			: INT; 						(* characteristic of the control algorithm for outlet port 4 -> choose characteristic from list *)

	//tuning parameters
		iOptProportionalGainFor2	: INT;						// Optional tuning parameter for the customized proportional element of the PID modulator at outlet port 2 [1 digit = 0.01 g/s/bar]
		iOptIntegralGainFor2		: INT;						// Optional tuning parameter for the customized integral element of the PID modulator at outlet port 2 [1 digit = 0.01 g/s²/bar]
		iOptTimeConstantFor2		: INT;						// Optional tuning parameter for the customized time constant element of the PID modulator at outlet port 2 [1 digit = 0.001 s]
		iOptProportionalGainFor4	: INT;						// Optional tuning parameter for the customized proportional element of the PID modulator at outlet port 4 [1 digit = 0.01 g/s/bar]
		iOptIntegralGainFor4		: INT;						// Optional tuning parameter for the customized integral element of the PID modulator at outlet port 4 [1 digit = 0.01 g/s²/bar]
		iOptTimeConstantFor4		: INT;						// Optional tuning parameter for the customized time constant element of the PID modulator at outlet port 4 [1 digit = 0.001 s]
END_VAR                     		

VAR_OUTPUT                  		
	iResponse 						: eTransferResponse; 		(* returns the status of the execution of the download process *)
	sCurrentValue 					: STRING; 					(* indicates which value of the array is currently treated (necessary to evaluate in case of error messages) *)
	xDownloadDone 					: BOOL; 					(* indicates whether the download was successful *)
	xDownloadError 					: BOOL := FALSE; 			(* indicates whether an error occurred during the transfer *)
END_VAR                     		

VAR                         		
	aTransferPackages				: ARRAY [0..100] OF stTransferPackage;
	fbdownloadMultipleParameters	: FB_Download_Multiple_Parameters;
	iCurrentValue					: INT;
	fbWriteValueToWord 				: FB_Write_Value_To_Word;
END_VAR

(*****************************************************************************************************

Festo SE & Co. KG, Esslingen
Copyright (c) 2018. All rights reserved.

Product:            Motion Terminal VTEM
Description:        Function block to download the parameters for Motion App 3 to the Motion Terminal

Object version:     2.00
Last change:        2019-03
======================================================================================================
                                       H I S T O R Y
======================================================================================================
Version:            2.00
Date:               2019-03
Change/Activity:    - added parameters for the sensor port mapping (#2256294)
                    - changed awBusDataToVTEM into VAR_IN_OUT (#2368965)
Release:            3.5.7.230 (CODESYS 3.5.7.2, Lib version 3.0)
Author:             JEBU
------------------------------------------------------------------------------------------------------
Version:            1.01
Date:               2018-11
Change/Activity:    - added tuning parameters (#2257307)
Release:            3.5.7.221
Author:             JEBU
------------------------------------------------------------------------------------------------------
Version:            1.00
Date:               2017
Change/Activity:    - created
Release:            3.5.7.220
Author:             HLBG
======================================================================================================

*****************************************************************************************************)

// write the Motion App specific parameters into the struct
	//iCharacteristicAt2
		aTransferPackages[0].iChannel := iParameterSet;
		aTransferPackages[0].iAddressedTarget := 3;
		aTransferPackages[0].iIndex := 220;
		aTransferPackages[0].iTransferValue := iCharacteristicAt2;
	
	//iCharacteristicAt4
		aTransferPackages[1].iChannel := iParameterSet;
		aTransferPackages[1].iAddressedTarget := 3;
		aTransferPackages[1].iIndex := 221;
		aTransferPackages[1].iTransferValue := iCharacteristicAt4;
	
	//iOptProportionalGainFor2
		aTransferPackages[2].iChannel := iParameterSet;
		aTransferPackages[2].iAddressedTarget := 3;
		aTransferPackages[2].iIndex := 230;
		aTransferPackages[2].iTransferValue := iOptProportionalGainFor2;
		
	//iOptIntegralGainFor2
		aTransferPackages[3].iChannel := iParameterSet;
		aTransferPackages[3].iAddressedTarget := 3;
		aTransferPackages[3].iIndex := 231;
		aTransferPackages[3].iTransferValue := iOptIntegralGainFor2;
		
	//iOptTimeConstantFor2
		aTransferPackages[4].iChannel := iParameterSet;
		aTransferPackages[4].iAddressedTarget := 3;
		aTransferPackages[4].iIndex := 232;
		aTransferPackages[4].iTransferValue := iOptTimeConstantFor2;
		
	//iOptProportionalGainFor4
		aTransferPackages[5].iChannel := iParameterSet;
		aTransferPackages[5].iAddressedTarget := 3;
		aTransferPackages[5].iIndex := 240;
		aTransferPackages[5].iTransferValue := iOptProportionalGainFor4;
		
	//iOptIntegralGainFor4
		aTransferPackages[6].iChannel := iParameterSet;
		aTransferPackages[6].iAddressedTarget := 3;
		aTransferPackages[6].iIndex := 241;
		aTransferPackages[6].iTransferValue := iOptIntegralGainFor4;
		
	//iOptTimeConstantFor4
		aTransferPackages[7].iChannel := iParameterSet;
		aTransferPackages[7].iAddressedTarget := 3;
		aTransferPackages[7].iIndex := 242;
		aTransferPackages[7].iTransferValue := iOptTimeConstantFor4;
	
	//iInPortRetract_optional
		aTransferPackages[8].iChannel := iParameterSet;
		aTransferPackages[8].iAddressedTarget := 3;
		aTransferPackages[8].iIndex := 70;
		aTransferPackages[8].iTransferValue := iInPortRetracted_optional;
	
	//iInPortAdvanced_optional
		aTransferPackages[9].iChannel := iParameterSet;
		aTransferPackages[9].iAddressedTarget := 3;
		aTransferPackages[9].iIndex := 71;
		aTransferPackages[9].iTransferValue := iInPortAdvanced_optional;
		
	// define end of parameter list to be downloaded by setting all variables to 0 (end criterion for FB_Download_Multiple_Parameters)
		aTransferPackages[10].iChannel := 0;
		aTransferPackages[10].iAddressedTarget := 0;
		aTransferPackages[10].iIndex := 0;
		aTransferPackages[10].iTransferValue := 0;

// pre-check of the value for the parameter set
	IF xExecute = TRUE AND (iParameterSet < 1 OR iParameterSet > 5) THEN		// invalid input for the parameter set
		xDownloadDone := FALSE; 
		xDownloadError := TRUE; 
		iResponse := eTransferResponse.invalid_ParameterSet; 
		iCurrentValue := 0; 
		// send command 'stop'
		fbWriteValueToWord(iValue := 61, iStartBit := 0, iEndBit := 5, wDataWord := awBusDataToVTEM[0]); 			// ValveMode = 61
		fbWriteValueToWord(iValue := 0, iStartBit := 6, iEndBit := 15, wDataWord := awBusDataToVTEM[0]); 			// (empty)
		awBusDataToVTEM[1] := 0; 
		awBusDataToVTEM[2] := 0; 
		
	ELSE	
		// call the function block for multiple parameter download
			fbdownloadMultipleParameters(	xExecute := xExecute,
											awBusDataFromVTEM := awBusDataFromVTEM,
											aTransferPackages := aTransferPackages, 
											awBusDataToVTEM := awBusDataToVTEM,
											xDownloadDone => xDownloadDone,
											xDownloadError => xDownloadError,
											iResponse => iResponse,
											iCurrentValue => iCurrentValue);
	END_IF


// The current value output is needed if there is any invalid value in order to address it correctly.
// As the user doesn't work with indices in this function block, the current value is transformed to a string holding the name of the parameter.
	CASE iCurrentValue OF
		0: sCurrentValue := 'iCharacteristicAt2';
		1: sCurrentValue := 'iCharacteristicAt4';
		2: sCurrentValue := 'iOptProportionalGainFor2';
		3: sCurrentValue := 'iOptIntegralGainFor2';
		4: sCurrentValue := 'iOptTimeConstantFor2';
		5: sCurrentValue := 'iOptProportionalGainFor4';
		6: sCurrentValue := 'iOptIntegralGainFor4';
		7: sCurrentValue := 'iOptTimeConstantFor4';
		8: sCurrentValue := 'iInPortRetract_optional';
		9: sCurrentValue := 'iInPortAdvanced_optional';
		10: sCurrentValue := 'AllParametersWritten';
	END_CASE

END_FUNCTION_BLOCK

// Transfermode/specific_MA_config/FB_Write_config_MA_08
/// This function block can be used to download the configuration of Motion App 8 ("Selectable pressure level (ECO)").
/// The specific parameters of this Motion App are the inputs of this FB and can be defined by the user. 
/// The function block uses the transfer mode to write this configuration to the Motion Terminal
/// and indicates the state of the download process.

FUNCTION_BLOCK FB_Write_config_MA_08
VAR_INPUT
	awBusDataFromVTEM 				: ARRAY [0..2] OF WORD;		(* 6 bytes of process data received from the Motion Terminal *)
END_VAR

VAR_IN_OUT
	awBusDataToVTEM 				: ARRAY [0..2] OF WORD; 	(* 6 bytes of process data sent to the Motion Terminal *)
END_VAR

VAR_INPUT
	xExecute 						: BOOL; 					(* has to be set to TRUE for a download and to FALSE to reset the function block after a download *)
		                    		                        	
	iParameterSet					: INT := 1; 				(* the parameter set to be written to, 1 by default *)
	
	// system parameters
		iTubingLengthAt2 			: INT; 						(* length of the tubing connected to outlet port 2 of the valve [1 digit = 1 mm] *)
	 	iTubingLengthAt4 			: INT;						(* length of the tubing connected to outlet port 4 of the valve [1 digit = 1 mm] *)
	 	iTubingInnerDiameterAt2		: INT;  					(* inner diameter of the tubing connected to outlet port 2 of the valve [1 digit = 0.01 mm] *)
	 	iTubingInnerDiameterAt4		: INT;						(* inner diameter of the tubing connected to outlet port 4 of the valve [1 digit = 0.01 mm] *)
	 	iDriveType 					: INT;						(* type of the drive/cylinder/... that is to be operated by the valve ->  see list of drive types *)
	 	iDriveStroke 				: INT; 						(* stroke of the drive/cylinder/... that is to be operated by the valve [1 digit = 1mm for linear drives, 1 digit = 1° for rotary drives] *)
		iInstallationPositionDrive 	: INT;  	 				(* inclination of the cylinder with reference to a horizontal installation position [1 digit = 0.01°, positive values = advancing upwards] *)
		iInPortRetracted_optional	: INT;						// Sensor port for detection of end position at pressurisation of outlet port 2 (retracted), value is number of the slot (beginning from 0) * 10 + number of the port
		iInPortAdvanced_optional	: INT;						// Sensor port for detection of end position at pressurisation of outlet port 4 (advanced), value is number of the slot (beginning from 0) * 10 + number of the port
	
	// application parameters                               	
		iLoadRetracting 			: INT;						(* mass that is to be moved by the drive when retracting ((2) pressurised) [1 digit = 0.01 kg] *)
	 	iLoadAdvancing 				: INT; 						(* mass that is to be moved by the drive when advancing ((4) pressurised) [1 digit = 0.01 kg] *)
		iMomentOfInertiaRetracting	: INT;						// Moment of inertia during for swivel drives when retratcting ((2) pressirised) [1 digit = 1 kg cm³]
		iMomentOfInertiaAdvancing	: INT;						// Moment of inertia during for swivel drives when advancing ((4) pressirised) [1 digit = 1 kg cm³]
		iSoftStartFunction			: INT := 1;					(* flag to enable or disable the iSoftStartFunction; 0 = disabled, 1 = enabled *)
END_VAR

VAR_OUTPUT                                                  	
	iResponse 						: eTransferResponse; 		(* returns the status of the execution of the download process *)
	sCurrentValue 					: STRING; 					(* indicates which value of the array is currently treated (necessary to evaluate in case of error messages) *)
	xDownloadDone 					: BOOL; 					(* indicates whether the download was successful *)
	xDownloadError 					: BOOL := FALSE; 			(* indicates whether an error occurred during the transfer *)
END_VAR

VAR
	aTransferPackages				: ARRAY [0..100] OF stTransferPackage;
	fbdownloadMultipleParameters 	: FB_Download_Multiple_Parameters;
	iCurrentValue					: INT;
	fbWriteValueToWord 				: FB_Write_Value_To_Word;
END_VAR

(*****************************************************************************************************

Festo SE & Co. KG, Esslingen
Copyright (c) 2018. All rights reserved.

Product:            Motion Terminal VTEM
Description:        Function block to download the parameters for Motion App 8 to the Motion Terminal

Object version:     2.00
Last change:        2019-03
======================================================================================================
                                       H I S T O R Y
======================================================================================================
Version:            2.00
Date:               2019-03
Change/Activity:    - added parameters for moment of inertia used for swivel drives (#2307852)
                    - added parameters for the sensor port mapping (#2256294)
                    - changed awBusDataToVTEM into VAR_IN_OUT (#2368965)
Release:            3.5.7.230 (CODESYS 3.5.7.2, Lib version 3.0)
Author:             JEBU
------------------------------------------------------------------------------------------------------
Version:            1.00
Date:               2017
Change/Activity:    - created
Release:            3.5.7.220
Author:             HLBG
======================================================================================================

*****************************************************************************************************)

// write the Motion App specific parameters into the struct
	//iTubingLengthAt2
		aTransferPackages[0].iChannel := iParameterSet;
		aTransferPackages[0].iAddressedTarget := 8;
		aTransferPackages[0].iIndex := 12;
		aTransferPackages[0].iTransferValue := iTubingLengthAt2;
		
	//iTubingLengthAt4
		aTransferPackages[1].iChannel := iParameterSet;
		aTransferPackages[1].iAddressedTarget := 8;
		aTransferPackages[1].iIndex := 13;
		aTransferPackages[1].iTransferValue := iTubingLengthAt4;
		
	//iTubingInnerDiameterAt2
		aTransferPackages[2].iChannel := iParameterSet;
		aTransferPackages[2].iAddressedTarget := 8;
		aTransferPackages[2].iIndex := 14;
		aTransferPackages[2].iTransferValue := iTubingInnerDiameterAt2;
		
	//iTubingInnerDiameterAt4
		aTransferPackages[3].iChannel := iParameterSet;
		aTransferPackages[3].iAddressedTarget := 8;
		aTransferPackages[3].iIndex := 15;
		aTransferPackages[3].iTransferValue := iTubingInnerDiameterAt4;
		
	//iDriveType
		aTransferPackages[4].iChannel := iParameterSet;
		aTransferPackages[4].iAddressedTarget := 8;
		aTransferPackages[4].iIndex := 20;
		aTransferPackages[4].iTransferValue := iDriveType;
		
	//iDriveStroke
		aTransferPackages[5].iChannel := iParameterSet;
		aTransferPackages[5].iAddressedTarget := 8;
		aTransferPackages[5].iIndex := 21;
		aTransferPackages[5].iTransferValue := iDriveStroke;
		
	//iInstallationPositionDrive
		aTransferPackages[6].iChannel := iParameterSet;
		aTransferPackages[6].iAddressedTarget := 8;
		aTransferPackages[6].iIndex := 60;
		aTransferPackages[6].iTransferValue := iInstallationPositionDrive;
		
	//iLoadRetracting
		aTransferPackages[7].iChannel := iParameterSet;
		aTransferPackages[7].iAddressedTarget := 8;
		aTransferPackages[7].iIndex := 100;
		aTransferPackages[7].iTransferValue := iLoadRetracting;
		
	//iLoadAdvancing
		aTransferPackages[8].iChannel := iParameterSet;
		aTransferPackages[8].iAddressedTarget := 8;
		aTransferPackages[8].iIndex := 101;
		aTransferPackages[8].iTransferValue := iLoadAdvancing;
		
	//iMomentOfInertiaRetracting
		aTransferPackages[9].iChannel := iParameterSet;
		aTransferPackages[9].iAddressedTarget := 8;
		aTransferPackages[9].iIndex := 102;
		aTransferPackages[9].iTransferValue := iMomentOfInertiaRetracting;
	
	//iMomentOfInertiaAdvancing
		aTransferPackages[10].iChannel := iParameterSet;
		aTransferPackages[10].iAddressedTarget := 8;
		aTransferPackages[10].iIndex := 103;
		aTransferPackages[10].iTransferValue := iMomentOfInertiaAdvancing;

	//iSoftStartFunction
		aTransferPackages[11].iChannel := iParameterSet;
		aTransferPackages[11].iAddressedTarget := 8;
		aTransferPackages[11].iIndex := 222;
		aTransferPackages[11].iTransferValue := iSoftStartFunction;
		
	//iInPortRetract_optional
		aTransferPackages[12].iChannel := iParameterSet;
		aTransferPackages[12].iAddressedTarget := 8;
		aTransferPackages[12].iIndex := 70;
		aTransferPackages[12].iTransferValue := iInPortRetracted_optional;
	
	//iInPortAdvanced_optional
		aTransferPackages[13].iChannel := iParameterSet;
		aTransferPackages[13].iAddressedTarget := 8;
		aTransferPackages[13].iIndex := 71;
		aTransferPackages[13].iTransferValue := iInPortAdvanced_optional;
	
	// define end of parameter list to be downloaded by setting all variables to 0 (end criterion for FB_Download_Multiple_Parameters)
		aTransferPackages[14].iChannel := 0;
		aTransferPackages[14].iAddressedTarget := 0;
		aTransferPackages[14].iIndex := 0;
		aTransferPackages[14].iTransferValue := 0;


// pre-check of the value for the parameter set
	IF xExecute = TRUE AND (iParameterSet < 1 OR iParameterSet > 5) THEN		// invalid input for the parameter set
		xDownloadDone := FALSE; 
		xDownloadError := TRUE; 
		iResponse := eTransferResponse.invalid_ParameterSet; 
		iCurrentValue := 0; 
		// send command 'stop'
		fbWriteValueToWord(iValue := 61, iStartBit := 0, iEndBit := 5, wDataWord := awBusDataToVTEM[0]); 			// ValveMode = 61
		fbWriteValueToWord(iValue := 0, iStartBit := 6, iEndBit := 15, wDataWord := awBusDataToVTEM[0]); 			// (empty)
		awBusDataToVTEM[1] := 0; 
		awBusDataToVTEM[2] := 0; 
		
	ELSE	
		// call the function block for multiple parameter download
			fbdownloadMultipleParameters(	xExecute := xExecute,
											awBusDataFromVTEM := awBusDataFromVTEM,
											aTransferPackages := aTransferPackages, 
											awBusDataToVTEM := awBusDataToVTEM,
											xDownloadDone => xDownloadDone,
											xDownloadError => xDownloadError,
											iResponse => iResponse,
											iCurrentValue => iCurrentValue);
	END_IF


// The current value output is needed if there is any invalid value in order to address it correctly.
// As the user doesn't work with indices in this function block, the current value is transformed to a string holding the name of the parameter.
	CASE iCurrentValue OF
		0: sCurrentValue := 'iTubingLengthAt2';
		1: sCurrentValue := 'iTubingLengthAt4';
		2: sCurrentValue := 'iTubingInnerDiameterAt2';
		3: sCurrentValue := 'iTubingInnerDiameterAt4';
		4: sCurrentValue := 'iDriveType';
		5: sCurrentValue := 'iDriveStroke';
		6: sCurrentValue := 'iInstallationPositionDrive';
		7: sCurrentValue := 'iLoadRetracting';
		8: sCurrentValue := 'iLoadAdvancing';
		9: sCurrentValue := 'iMomentOfInertiaRetracting';
		10: sCurrentValue := 'iMomentOfInertiaAdvancing';
		11: sCurrentValue := 'iSoftStartFunction';
		12: sCurrentValue := 'iInPortRetract_optional';
		13: sCurrentValue := 'iInPortAdvanced_optional';
	  	14: sCurrentValue := 'AllParametersWritten';
	END_CASE

END_FUNCTION_BLOCK

// Transfermode/specific_MA_config/FB_Write_config_MA_05
/// This function block can be used to download the configuration of Motion App 5 ("Supply and exhaust air flow control").
/// The specific parameters of this Motion App are the inputs of this FB and can be defined by the user. 
/// The function block uses the transfer mode to write this configuration to the Motion Terminal
/// and indicates the state of the download process.

FUNCTION_BLOCK FB_Write_config_MA_05
VAR_INPUT
	awBusDataFromVTEM 				: ARRAY [0..2] OF WORD;		(* 6 bytes of process data received from the Motion Terminal *)
END_VAR

VAR_IN_OUT
	awBusDataToVTEM 				: ARRAY [0..2] OF WORD; 	(* 6 bytes of process data sent to the Motion Terminal *)
END_VAR

VAR_INPUT
	xExecute 						: BOOL; 					(* has to be set to TRUE for a download and to FALSE to reset the function block after a download *)
		                    		                        		
	iParameterSet					: INT := 1; 				(* the parameter set to be written to, 1 by default *)
                                                    		
	// system parameters
		iInPortRetracted_optional	: INT;						// Sensor port for detection of end position at pressurisation of outlet port 2 (retracted), value is number of the slot (beginning from 0) * 10 + number of the port
		iInPortAdvanced_optional	: INT;						// Sensor port for detection of end position at pressurisation of outlet port 4 (advanced), value is number of the slot (beginning from 0) * 10 + number of the port

	// application parameters                       	
		iSoftStartFunction			: INT := 1;					(* flag to enable or disable the iSoftStartFunction; 0 = disabled, 1 = enabled *)
END_VAR

VAR_OUTPUT
	iResponse 						: eTransferResponse; 		(* returns the status of the execution of the download process *)
	sCurrentValue 					: STRING; 					(* indicates which value of the array is currently treated (necessary to evaluate in case of error messages) *)
	xDownloadDone 					: BOOL; 					(* indicates whether the download was successful *)
	xDownloadError 					: BOOL := FALSE; 			(* indicates whether an error occurred during the transfer *)
END_VAR

VAR
	aTransferPackages				: ARRAY [0..100] OF stTransferPackage; 
	fbdownloadMultipleParameters 	: FB_Download_Multiple_Parameters; 
	iCurrentValue					: INT;
	fbWriteValueToWord 				: FB_Write_Value_To_Word; 
END_VAR

(*****************************************************************************************************

Festo SE & Co. KG, Esslingen
Copyright (c) 2018. All rights reserved.

Product:            Motion Terminal VTEM
Description:        Function block to download the parameters for Motion App 5 to the Motion Terminal

Object version:     2.00
Last change:        2019-03
======================================================================================================
                                       H I S T O R Y
======================================================================================================
Version:            2.00
Date:               2019-03
Change/Activity:    - added parameters for the sensor port mapping (#2256294)
                    - changed awBusDataToVTEM into VAR_IN_OUT (#2368965)
Release:            3.5.7.230 (CODESYS 3.5.7.2, Lib version 3.0)
Author:             JEBU
------------------------------------------------------------------------------------------------------
Version:            1.00
Date:               2017
Change/Activity:    - created
Release:            3.5.7.220
Author:             HLBG
======================================================================================================

*****************************************************************************************************)

// write the Motion App specific parameters into the struct
	//iSoftStartFunction
		aTransferPackages[0].iChannel := iParameterSet;
		aTransferPackages[0].iAddressedTarget := 5;
		aTransferPackages[0].iIndex := 222;
		aTransferPackages[0].iTransferValue := iSoftStartFunction;
	
	//iInPortRetract_optional
		aTransferPackages[1].iChannel := iParameterSet;
		aTransferPackages[1].iAddressedTarget := 5;
		aTransferPackages[1].iIndex := 70;
		aTransferPackages[1].iTransferValue := iInPortRetracted_optional;
	
	//iInPortAdvanced_optional
		aTransferPackages[2].iChannel := iParameterSet;
		aTransferPackages[2].iAddressedTarget := 5;
		aTransferPackages[2].iIndex := 71;
		aTransferPackages[2].iTransferValue := iInPortAdvanced_optional;
	
	// define end of parameter list to be downloaded by setting all variables to 0 (end criterion for FB_Download_Multiple_Parameters)
		aTransferPackages[3].iChannel := 0;
		aTransferPackages[3].iAddressedTarget := 0;
		aTransferPackages[3].iIndex := 0;
		aTransferPackages[3].iTransferValue := 0;


// pre-check of the value for the parameter set
	IF xExecute = TRUE AND (iParameterSet < 1 OR iParameterSet > 5) THEN		// invalid input for the parameter set
		xDownloadDone := FALSE; 
		xDownloadError := TRUE; 
		iResponse := eTransferResponse.invalid_ParameterSet; 
		iCurrentValue := 0; 
		// send command 'stop'
		fbWriteValueToWord(iValue := 61, iStartBit := 0, iEndBit := 5, wDataWord := awBusDataToVTEM[0]); 			// ValveMode = 61
		fbWriteValueToWord(iValue := 0, iStartBit := 6, iEndBit := 15, wDataWord := awBusDataToVTEM[0]); 			// (empty)
		awBusDataToVTEM[1] := 0; 
		awBusDataToVTEM[2] := 0; 
		
	ELSE	
		// call the function block for multiple parameter download
			fbdownloadMultipleParameters(	xExecute := xExecute,
											awBusDataFromVTEM := awBusDataFromVTEM,
											aTransferPackages := aTransferPackages, 
											awBusDataToVTEM := awBusDataToVTEM,
											xDownloadDone => xDownloadDone,
											xDownloadError => xDownloadError,
											iResponse => iResponse,
											iCurrentValue => iCurrentValue);
	END_IF


// The current value output is needed if there is any invalid value in order to address it correctly.
// As the user doesn't work with indices in this function block, the current value is transformed to a string holding the name of the parameter.
	CASE iCurrentValue OF
		0: sCurrentValue := 'iSoftStartFunction';
		1: sCurrentValue := 'iInPortRetract_optional';
		2: sCurrentValue := 'iInPortAdvanced_optional';
		3: sCurrentValue := 'AllParametersWritten';
	END_CASE

END_FUNCTION_BLOCK

// StateInterpreter/FB_StateInterpreter_MA_33
/// The variable "byActualAppState" is an output of the FB_ValveControl that is used differently in each Motion App.
/// This function block interprets the "AppState" output of the FB_ValveControl if Motion App 33 ("Positioning") is running.
/// The Motion App specific values are derived from the "byActualAppState".

FUNCTION_BLOCK FB_StateInterpreter_MA_33
VAR_INPUT
	byActualAppState 			: BYTE; 	// output of the FB_ValveControl
END_VAR
VAR_OUTPUT
	xRetractedEndPos			: BOOL;  	// indicates whether the retracted end position (outlet port 4 pressurised) was reached (<= 1 mm) 
	xAdvancedEndPos				: BOOL;  	// indicates whether the advanced end position (outlet port 4 pressurised) was reached (<= 1 mm) 
	xTargetPositionReached		: BOOL;  	// TRUE if the absolute deviation of the actual position from the setpoint position does not exceed the value defined in the "Tolerance for Target Position Reached" parameter for at least the duration defined in the "Damping time for Target Position Reached" parameter.  
	xOvershootInPlannedPath		: BOOL;		// TRUE if the planned path contains an overshoot over the target position
	xControlledStop				: BOOL;		// TRUE if a controlled stop was triggered by an end position violation (only active if the end position monitoring was not deactivated by the corresponding application parameter)
	xWarning					: BOOL; 	// indicates whether there is a warning returned by the Motion App
END_VAR
VAR
	fbReadBitsFromByte			: FB_Read_Bits_From_Byte;
	byRetractedEndPos			: BYTE;
	byAdvancedEndPos			: BYTE;
	byTargetPositionReached		: BYTE;
	byOvershootInPlannedPath	: BYTE;
	byControlledStop			: BYTE;      
	byWarning					: BYTE;
END_VAR

(*****************************************************************************************************

Festo SE & Co. KG, Esslingen
Copyright (c) 2019. All rights reserved.

Product:            Motion Terminal VTEM
Description:        Function block for interpreting the app state of Motion App 33 

Object version:     1.01
Last change:        2020-04
======================================================================================================
                                       H I S T O R Y
======================================================================================================
Version:            1.01
Date:               2020-04
Change/Activity:    - created (#2256322)
Release:            3.5.7.235 (CODESYS 3.5.7.2, Lib version 3.5)
Author:             JEBU
======================================================================================================

*****************************************************************************************************)

// read the Motion App specific values from the ActualAppState byte
fbReadBitsFromByte(byData := byActualAppState, iStartBit := 0, iEndBit := 0, byValue => byRetractedEndPos);
xRetractedEndPos :=  BYTE_TO_BIT(byRetractedEndPos);

fbReadBitsFromByte(byData := byActualAppState, iStartBit := 2, iEndBit := 2, byValue => byAdvancedEndPos); 
xAdvancedEndPos :=  BYTE_TO_BIT(byAdvancedEndPos);

fbReadBitsFromByte(byData := byActualAppState, iStartBit := 1, iEndBit := 1, byValue => byTargetPositionReached);
xTargetPositionReached :=  BYTE_TO_BIT(byTargetPositionReached);

fbReadBitsFromByte(byData := byActualAppState, iStartBit := 5, iEndBit := 5, byValue => byOvershootInPlannedPath);
xOvershootInPlannedPath :=  BYTE_TO_BIT(byOvershootInPlannedPath);

fbReadBitsFromByte(byData := byActualAppState, iStartBit := 6, iEndBit := 6, byValue => byControlledStop);
xControlledStop :=  BYTE_TO_BIT(byControlledStop);

fbReadBitsFromByte(byData := byActualAppState, iStartBit := 7, iEndBit := 7, byValue => byWarning);
xWarning := BYTE_TO_BIT(byWarning);

END_FUNCTION_BLOCK

// Transfermode/specific_MA_config/FB_Write_config_MA_01
/// This function block can be used to download the configuration of Motion App 1 ("Proportional directional control valve").
/// The specific parameters of this Motion App are the inputs of this FB and can be defined by the user. 
/// The function block uses the transfer mode to write this configuration to the Motion Terminal
/// and indicates the state of the download process.

FUNCTION_BLOCK FB_Write_config_MA_01
VAR_INPUT
	awBusDataFromVTEM 				: ARRAY [0..2] OF WORD;		(* 6 bytes of process data received from the Motion Terminal *)
END_VAR
	
VAR_IN_OUT
	awBusDataToVTEM 				: ARRAY [0..2] OF WORD; 	(* 6 bytes of process data sent to the Motion Terminal *)
END_VAR

VAR_INPUT
	xExecute 						: BOOL; 					(* has to be set to TRUE for a download and to FALSE to reset the function block after a download *)

	iParameterSet					: INT := 1; 				(* the parameter set to be written to, 1 by default *)
	
	// system parameters
		iInPortRetracted_optional	: INT;						// Sensor port for detection of end position at pressurisation of outlet port 2 (retracted), value is number of the slot (beginning from 0) * 10 + number of the port
		iInPortAdvanced_optional	: INT;						// Sensor port for detection of end position at pressurisation of outlet port 4 (advanced), value is number of the slot (beginning from 0) * 10 + number of the port

	// application parameters
		iOperatingMode				: INT := 0;	 				// Switching the operating mode between open-loop controlled (0) and close-loop controlled (1) 
END_VAR                     		

VAR_OUTPUT                  		
	iResponse 						: eTransferResponse; 		(* returns the status of the execution of the download process *)
	sCurrentValue 					: STRING; 					(* indicates which value of the array is currently treated (necessary to evaluate in case of error messages) *)
	xDownloadDone 					: BOOL; 					(* indicates whether the download was successful *)
	xDownloadError 					: BOOL := FALSE; 			(* indicates whether an error occurred during the transfer *)
END_VAR

VAR
	aTransferPackages				: ARRAY [0..100] OF stTransferPackage;
	fbdownloadMultipleParameters 	: FB_Download_Multiple_Parameters;
	iCurrentValue					: INT;
	fbWriteValueToWord 				: FB_Write_Value_To_Word;
END_VAR

(*****************************************************************************************************

Festo SE & Co. KG, Esslingen
Copyright (c) 2018. All rights reserved.

Product:            Motion Terminal VTEM
Description:        Function Block to download the parameters for Motion App 1 to the Motion Terminal

Object version:     2.00
Last change:        2019-03
======================================================================================================
                                       H I S T O R Y
======================================================================================================
Version:            2.00
Date:               2019-03
Change/Activity:    - created (#2256983)
Release:            3.5.7.230 (CODESYS 3.5.7.2, Lib version 3.0)
Author:             JEBU
======================================================================================================

*****************************************************************************************************)

// write the Motion App specific parameters into the struct
	//iOperatingMode
		aTransferPackages[0].iChannel := iParameterSet;
		aTransferPackages[0].iAddressedTarget := 1;
		aTransferPackages[0].iIndex := 223;
		aTransferPackages[0].iTransferValue := iOperatingMode;
	
	//iInPortRetract_optional
		aTransferPackages[1].iChannel := iParameterSet;
		aTransferPackages[1].iAddressedTarget := 1;
		aTransferPackages[1].iIndex := 70;
		aTransferPackages[1].iTransferValue := iInPortRetracted_optional;
	
	//iInPortRetract_optional
		aTransferPackages[2].iChannel := iParameterSet;
		aTransferPackages[2].iAddressedTarget := 1;
		aTransferPackages[2].iIndex := 71;
		aTransferPackages[2].iTransferValue := iInPortAdvanced_optional;
	
	// define end of parameter list to be downloaded by setting all variables to 0 (end criterion for FB_Download_Multiple_Parameters)
		aTransferPackages[3].iChannel := 0;
		aTransferPackages[3].iAddressedTarget := 0;
		aTransferPackages[3].iIndex := 0;
		aTransferPackages[3].iTransferValue := 0;


// pre-check of the value for the parameter set
	IF xExecute = TRUE AND (iParameterSet < 1 OR iParameterSet > 5) THEN		// invalid input for the parameter set
		xDownloadDone := FALSE; 
		xDownloadError := TRUE; 
		iResponse := eTransferResponse.invalid_ParameterSet; 
		iCurrentValue := 0; 
		// send command 'stop'
		fbWriteValueToWord(iValue := 61, iStartBit := 0, iEndBit := 5, wDataWord := awBusDataToVTEM[0]); 			// ValveMode = 61
		fbWriteValueToWord(iValue := 0, iStartBit := 6, iEndBit := 15, wDataWord := awBusDataToVTEM[0]); 			// (empty)
		awBusDataToVTEM[1] := 0; 
		awBusDataToVTEM[2] := 0; 
		
	ELSE	
		// call the function block for multiple parameter download
		fbdownloadMultipleParameters(	xExecute := xExecute,
										awBusDataFromVTEM := awBusDataFromVTEM,
										aTransferPackages := aTransferPackages, 
										awBusDataToVTEM := awBusDataToVTEM,
										xDownloadDone => xDownloadDone,
										xDownloadError => xDownloadError,
										iResponse => iResponse,
										iCurrentValue => iCurrentValue);
	END_IF
	
	
// The current value output is needed if there is any invalid value in order to address it correctly.
// As the user doesn't work with indices in this function block, the current value is transformed to a string holding the name of the parameter.
	CASE iCurrentValue OF
		0: sCurrentValue := 'iOperatingMode';
		1: sCurrentValue := 'iInPortRetract_optional';
		2: sCurrentValue := 'iInPortAdvanced_optional';
		3: sCurrentValue := 'AllParametersWritten';
	END_CASE

END_FUNCTION_BLOCK

// Transfermode/specific_MA_config/FB_Write_config_MA_06
/// This function block can be used to download the configuration of Motion App 6 ("ECO_drive").
/// The specific parameters of this Motion App are the inputs of this FB and can be defined by the user. 
/// The function block uses the transfer mode to write this configuration to the Motion Terminal
/// and indicates the state of the download process.

FUNCTION_BLOCK FB_Write_config_MA_06
VAR_INPUT
	awBusDataFromVTEM 				: ARRAY [0..2] OF WORD;		(* 6 bytes of process data received from the Motion Terminal *)
END_VAR
	
VAR_IN_OUT
	awBusDataToVTEM 				: ARRAY [0..2] OF WORD; 	(* 6 bytes of process data sent to the Motion Terminal *)
END_VAR

VAR_INPUT
	xExecute 						: BOOL; 					(* has to be set to TRUE for a download and to FALSE to reset the function block after a download *)

	iParameterSet					: INT := 1; 				(* the parameter set to be written to, 1 by default *)
	
	// system parameters
		iInPortRetracted			: INT;						// Sensor port for detection of end position at pressurisation of outlet port 2 (retracted), value is number of the slot (beginning from 0) * 10 + number of the port
		iInPortAdvanced				: INT;						// Sensor port for detection of end position at pressurisation of outlet port 4 (advanced), value is number of the slot (beginning from 0) * 10 + number of the port

END_VAR

VAR_OUTPUT                  		
	iResponse 						: eTransferResponse; 		(* returns the status of the execution of the download process *)
	sCurrentValue 					: STRING; 					(* indicates which value of the array is currently treated (necessary to evaluate in case of error messages) *)
	xDownloadDone 					: BOOL; 					(* indicates whether the download was successful *)
	xDownloadError 					: BOOL := FALSE; 			(* indicates whether an error occurred during the transfer *)
END_VAR

VAR
	aTransferPackages				: ARRAY [0..100] OF stTransferPackage;
	fbdownloadMultipleParameters 	: FB_Download_Multiple_Parameters;
	iCurrentValue					: INT;
	fbWriteValueToWord 				: FB_Write_Value_To_Word;
END_VAR

(*****************************************************************************************************

Festo SE & Co. KG, Esslingen
Copyright (c) 2018. All rights reserved.

Product:            Motion Terminal VTEM
Description:        Function Block to download the parameters for Motion App 6 to the Motion Terminal

Object version:     2.00
Last change:        2019-03
======================================================================================================
                                       H I S T O R Y
======================================================================================================
Version:            2.00
Date:               2019-03
Change/Activity:    - created (#2368895)
Release:            3.5.7.230 (CODESYS 3.5.7.2, Lib version 3.0)
Author:             JEBU
======================================================================================================

*****************************************************************************************************)

// write the Motion App specific parameters into the struct
	//iInPortRetract
		aTransferPackages[0].iChannel := iParameterSet;
		aTransferPackages[0].iAddressedTarget := 6;
		aTransferPackages[0].iIndex := 70;
		aTransferPackages[0].iTransferValue := iInPortRetracted;
	
	//iInPortRetract
		aTransferPackages[1].iChannel := iParameterSet;
		aTransferPackages[1].iAddressedTarget := 6;
		aTransferPackages[1].iIndex := 71;
		aTransferPackages[1].iTransferValue := iInPortAdvanced;
	
	// define end of parameter list to be downloaded by setting all variables to 0 (end criterion for FB_Download_Multiple_Parameters)
		aTransferPackages[2].iChannel := 0;
		aTransferPackages[2].iAddressedTarget := 0;
		aTransferPackages[2].iIndex := 0;
		aTransferPackages[2].iTransferValue := 0;


// pre-check of the value for the parameter set
	IF xExecute = TRUE AND (iParameterSet < 1 OR iParameterSet > 5) THEN		// invalid input for the parameter set
		xDownloadDone := FALSE; 
		xDownloadError := TRUE; 
		iResponse := eTransferResponse.invalid_ParameterSet; 
		iCurrentValue := 0; 
		// send command 'stop'
		fbWriteValueToWord(iValue := 61, iStartBit := 0, iEndBit := 5, wDataWord := awBusDataToVTEM[0]); 			// ValveMode = 61
		fbWriteValueToWord(iValue := 0, iStartBit := 6, iEndBit := 15, wDataWord := awBusDataToVTEM[0]); 			// (empty)
		awBusDataToVTEM[1] := 0; 
		awBusDataToVTEM[2] := 0; 
		
	ELSE	
		// call the function block for multiple parameter download
			fbdownloadMultipleParameters(	xExecute := xExecute,
											awBusDataFromVTEM := awBusDataFromVTEM,
											aTransferPackages := aTransferPackages, 
											awBusDataToVTEM := awBusDataToVTEM,
											xDownloadDone => xDownloadDone,
											xDownloadError => xDownloadError,
											iResponse => iResponse,
											iCurrentValue => iCurrentValue);
	END_IF
	
	
// The current value output is needed if there is any invalid value in order to address it correctly.
// As the user doesn't work with indices in this function block, the current value is transformed to a string holding the name of the parameter.
	CASE iCurrentValue OF
		0: sCurrentValue := 'iInPortRetract';
		1: sCurrentValue := 'iInPortAdvanced';
		2: sCurrentValue := 'AllParametersWritten';
	END_CASE

END_FUNCTION_BLOCK

// Operation/FB_TeachInRun
/// This function block is designed to execute the teach-in run (Valve Mode 60) on a valve. 
/// Before executing the transfer mode, the Parameter 255 (Motion App to be tought in) is
/// parameterised with the value on the corresponding input.
/// After that the teach-in run is started and can be controlled via the input "iManualControl"
/// if the manual operation is possible for the selectes Motion App.

FUNCTION_BLOCK FB_TeachInRun
VAR_INPUT
	awBusDataFromVTEM				: ARRAY [0..2] OF WORD;				// 6 bytes of process data that is received from the Motion Terminal
END_VAR

VAR_IN_OUT
	awBusDataToVTEM					: ARRAY [0..2] OF WORD;				// 6 bytes of process data that is sent to the Motion Terminal
END_VAR

VAR_INPUT
	xEnable							: BOOL;								// has to be set to TRUE in order to operate the teach-in run on the valve, otherwise the teach-in run is stopped  
	iParameterSet					: INT;								// Parameter Set to be used for soring the learning data 
	iMotionAppToBeToughtIn			: INT;								// ID of the Motion App that is to be taught-in
	iOperatingMode					: INT;								// Sets operating mode of teach-in run (0 = Stop, 1 = Auto, 2 = Manual (only Motion App #11)
	iManualControl					: INT;								// Control input for manual execution of teach-in run (0 = Block, 1 = Advance, 2 = Retract, 3 = Exhaust)
	xAcknowledge					: BOOL;								// errors can be acknowledged (after they got inactive) with a rising edge at this input, while the FB is enabled
END_VAR

VAR_OUTPUT
	xDone							: BOOL;								// indicates that the teach-in run was finished successfully
	xError							: BOOL;								// indicates that an Error occured
	iResponse						: eResponseTeachInRun;				// returns the status of the TeachInRun function block
	sResponseDescription			: STRING;							// returns the status of the TeachInRun function block as string
	xWarning						: BOOL;								// indicates whether there is a warning returned by the teach-in run
	xRetractedEndPos_optional		: BOOL;								// only if digital sensors are installed (optional): indicates whether the retracted end position was reached (after outlet port 2 is pressurised)
	xAdvancedEndPos_optional		: BOOL;								// only if digital sensors are installed (optional): indicates whether the advanced end position was reached (after outlet port 4 is pressurised)
END_VAR

VAR
	// State machine variables
		iState						: INT := 10;						// Value for the local state machine
		xStateChange				: BOOL;								// TRUE if the state is to be changed
		iCommandNumber				: INT;								// Value for the command case

	// First Cycle variables
		iParameterSetFC				: INT;								// Variable to store value from first cycle
		iMotionAppToBeToughtInFC	: INT;								// Variable to store value from first cycle
		iOperatingModeFCC			: INT;								// Variable to store value from first cycle in state "Completed" or "Error"
		iManualControlFCC			: INT;								// Variable to store value from first cycle in state "Completed" or "Error"

	// Function block instances
		fbreadbitsfromword				: FB_Read_Bits_From_Word;			// 
		fbwritevaluetoword				: FB_Write_Value_To_Word;			//
		fbstateinterpreterteachinrun	: FB_StateInterpreter_TeachInRun;	//

	// Current Valve variables
		iCurrentValveMode			: INT;								// 
		iCurrentValveState			: INT;								//
		iCurrentAppState			: INT;								//
		iCurrentChannelTM			: INT;								//
		iCurrentAddressedTargetTM	: INT;								//
		iCurrentIndexTM				: INT;								//
		iCurrentValueTM				: INT;								//
		iCurrentTransferControlTM	: INT;								//
		
	// Misc variables
		xInputValid					: BOOL;								// TRUE if the values iParameterSet, iMotionAppToBeToughtIn and iOperatingMode are within valid range
		xInputConsistent			: BOOL;
		xInvalidCommand				: BOOL;
		iInvalidCommand				: INT;
		xNoValve					: BOOL;
		xWebConfigAccess			: BOOL;
		xInvalidMotionApp			: BOOL;
		
		xAcknowledgeLastCycle		: BOOL;
		
		xAcknowledgeCompleted		: BOOL;
		xReadyToComplete			: BOOL;
		xStateFinished				: BOOL;
		xStateError					: BOOL;
		
		iReadParameterSet			: INT;
		iWriteParameterSet			: INT;
		xReturnReadParameterSet		: BOOL;
		
		iCounter					: INT;
		iCounterMax					: INT := 3000;
		
		xTeachInRunWasActive		: BOOL;
END_VAR

(*****************************************************************************************************

Festo SE & Co. KG, Esslingen
Copyright (c) 2019. All rights reserved.

Product:            Motion Terminal VTEM
Description:        Function block to execute the teach-in run

Object version:     1.04
Last change:        2020-05
======================================================================================================
                                       H I S T O R Y
======================================================================================================
Version:            1.04 
Date:               2020-05        
Change/Activity:    - created (#2256363)
Release:            3.5.7.234
Author:             JEBU/MKLP
======================================================================================================

******************************************************************************************************)

// Read the current status of the the motion terminal
	fbreadbitsfromword(wData:= awBusDataFromVTEM[0], iStartBit:=0, iEndBit:= 5, iValue=> iCurrentValveMode, xError=> );						// read current valve mode
	fbreadbitsfromword(wData:= awBusDataFromVTEM[0], iStartBit:=6, iEndBit:= 7, iValue=> iCurrentValveState, xError=> );					// read current valve state

	IF iCurrentValveMode <> 63 THEN																										// Operating mode:
		fbreadbitsfromword(wData:= awBusDataFromVTEM[0], iStartBit:=8, iEndBit:= 15, iValue=> iCurrentAppState, xError=>);					// read app state
	ELSIF iCurrentValveMode = 63 THEN																									// Transfer mode:
		fbreadbitsfromword(wData:= awBusDataFromVTEM[0], iStartBit:= 8, iEndBit:= 12, iValue=> iCurrentChannelTM, xError=> );				// read current channel
		fbreadbitsfromword(wData:= awBusDataFromVTEM[0], iStartBit:= 13, iEndBit:= 15, iValue=> iCurrentTransferControlTM, xError=> );		// read current transfer control
		fbreadbitsfromword(wData:= awBusDataFromVTEM[1], iStartBit:= 0, iEndBit:= 7, iValue=> iCurrentAddressedTargetTM, xError=> );		// read current addressed target
		fbreadbitsfromword(wData:= awBusDataFromVTEM[1], iStartBit:= 8, iEndBit:= 15, iValue=> iCurrentIndexTM, xError=> );					// read current index
		fbreadbitsfromword(wData:= awBusDataFromVTEM[2], iStartBit:= 0, iEndBit:= 15, iValue=> iCurrentValueTM, xError=> );					// read current value
	END_IF
	
	IF iCurrentValveMode = 60 AND iState = 40 THEN
		fbstateinterpreterteachinrun.byActualAppState := INT_TO_BYTE(iCurrentAppState);
		
		fbstateinterpreterteachinrun();
				
		xRetractedEndPos_optional := fbstateinterpreterteachinrun.xRetractedEndPos_optional;
		xAdvancedEndPos_optional := fbstateinterpreterteachinrun.xAdvancedEndPos_optional;
		xWarning := fbstateinterpreterteachinrun.xWarning;
		iResponse := fbstateinterpreterteachinrun.iTeachInRunState;
	END_IF
//-----------------------------------------------------------------------------------------------------------

// Transition for RESETTING 
	IF xEnable = FALSE AND iState <> 10 AND iState <> 100 THEN
		xStateChange := TRUE;
		iState := 100;
	END_IF
//-----------------------------------------------------------------------------------------------------------

// Transition for WebConfig Access denied
	IF 	xWebConfigAccess = FALSE AND 
		xEnable = TRUE AND iState <> 10 AND 
		iCurrentValveMode = 61 AND iCurrentAppState = 10 THEN 	// The WebConfig has write permission -> access denied for the PLC
			xStateChange := TRUE;
			iState := 70;
			xWebConfigAccess := TRUE;
	END_IF
//-----------------------------------------------------------------------------------------------------------
	
// Check if input data is consisent (not in state 10 IDLE)
	IF 	xInputConsistent = TRUE  AND 
		xEnable = TRUE AND iState <> 10 AND iState <> 15 AND 
		(iParameterSet <> iParameterSetFC OR iMotionAppToBeToughtIn <> iMotionAppToBeToughtInFC OR (iState = 70 AND xStateChange = FALSE AND (iOperatingModeFCC <> iOperatingMode OR iManualControlFCC <> iManualControl))) THEN
			xStateChange := TRUE;
			iState := 70;		// Input data inconsistent
			xInputConsistent := FALSE;		
	END_IF
	
	IF xNoValve = FALSE AND 
	   xEnable = TRUE AND iState <> 10 AND iState <> 15 AND 
	   iCurrentValveMode = 61 AND iCurrentValveState = 1 AND iCurrentAppState = 15 THEN		// no Valve detected 
			xNoValve := TRUE;
			xStateChange := TRUE;
			iState := 70;
	END_IF
//-----------------------------------------------------------------------------------------------------------

// Local state machine
	CASE iState OF
		10:	// IDLE mode
			// code that is executed only in the first cycle of this state
				IF xStateChange = TRUE THEN
					xStateChange := FALSE;
				END_IF
			//-----------------------------------------------------------------------------------------------------------
			
			// code that is repeated every cycle in this state	
				iCommandNumber := 0;	// IDLE
				iResponse := eResponseTeachInRun.idle;
			//-----------------------------------------------------------------------------------------------------------
			
			// Transition
				IF xEnable = TRUE THEN
					xStateChange := TRUE;	// Leave this state
					iState := 15;
				END_IF
			//-----------------------------------------------------------------------------------------------------------

